(* IEC 61131-3 sources: RL_MAR/experiments/comparison/llm4plc/results/gpt-4o_20260507_114630/20260507_121514, 1 file *)

(* ---- generated_code_iteration_0.st ---- *)
plaintext
START_ST
FUNCTION_BLOCK TrafficManagementSystem
VAR_INPUT
    VehicleCount1 : INT; (* Input for vehicle count at intersection 1 *)
    VehicleCount2 : INT; (* Input for vehicle count at intersection 2 *)
    VehicleCount3 : INT; (* Input for vehicle count at intersection 3 *)
    VehicleCount4 : INT; (* Input for vehicle count at intersection 4 *)
END_VAR
VAR_OUTPUT
    TrafficLight1 : BOOL; (* Output for traffic light at intersection 1 *)
    TrafficLight2 : BOOL; (* Output for traffic light at intersection 2 *)
    TrafficLight3 : BOOL; (* Output for traffic light at intersection 3 *)
    TrafficLight4 : BOOL; (* Output for traffic light at intersection 4 *)
END_VAR
VAR
    state : INT := 0; (* State variable to track the current state of the FSM *)
    prevState : INT := -1; (* Previous state variable to track the last state *)
END_VAR

(* FSM Logic *)
CASE state OF
    (* STATE 0: Initialize all traffic lights to red (FALSE) *)
    0:
        TrafficLight1 := FALSE;
        TrafficLight2 := FALSE;
        TrafficLight3 := FALSE;
        TrafficLight4 := FALSE;
        state := 1; (* Transition to STATE 1 *)

    (* STATE 1: Evaluate intersections 1 and 2 *)
    1:
        IF VehicleCount1 > VehicleCount2 THEN
            TrafficLight1 := TRUE;
            TrafficLight2 := FALSE;
        ELSIF VehicleCount2 > VehicleCount1 THEN
            TrafficLight1 := FALSE;
            TrafficLight2 := TRUE;
        ELSE
            TrafficLight1 := FALSE; (* Default to red if counts are equal *)
            TrafficLight2 := FALSE;
        END_IF;
        state := 2; (* Transition to STATE 2 *)

    (* STATE 2: Evaluate intersections 3 and 4 *)
    2:
        IF VehicleCount3 > VehicleCount4 THEN
            TrafficLight3 := TRUE;
            TrafficLight4 := FALSE;
        ELSIF VehicleCount4 > VehicleCount3 THEN
            TrafficLight3 := FALSE;
            TrafficLight4 := TRUE;
        ELSE
            TrafficLight3 := FALSE; (* Default to red if counts are equal *)
            TrafficLight4 := FALSE;
        END_IF;
        state := 1; (* Transition back to STATE 1 *)

    (* Default case to handle unexpected states *)
    ELSE
        state := 0; (* Reset to STATE 0 in case of an invalid state *)
END_CASE;

END_FUNCTION_BLOCK
END_ST
